// TwinCAT 3 PLC project PLC1
// ProgramVersion: 3.1.4024.0
// libraries:
//   Tc2_Standard, * (Beckhoff Automation GmbH)
//   Tc2_System, * (Beckhoff Automation GmbH)
//   Tc3_Module, * (Beckhoff Automation GmbH)
// project tree:
//   / PlcTask.TcTTO
//   POUs/ FB_ParseString.TcPOU, MAIN.TcPOU
// real-time tasks:
//   TASK PlcTask: cycle T#10ms, priority 20, ADS port 350

CONFIGURATION PLC1
    RESOURCE PLC ON TwinCAT3
        TASK PlcTask(INTERVAL := T#10ms, PRIORITY := 20);
        PROGRAM MAIN WITH PlcTask : MAIN;
    END_RESOURCE
END_CONFIGURATION

// ---- POUs/MAIN.TcPOU
PROGRAM MAIN
VAR
END_VAR

END_PROGRAM

// ---- POUs/FB_ParseString.TcPOU
FUNCTION_BLOCK FB_ParseString
VAR_INPUT
	sCharToSearch : STRING;
	sInputString  : STRING;
END_VAR
VAR_OUTPUT
	sStringParsed : STRING;
END_VAR
VAR
	Position: INT;
END_VAR

Position := FIND(sInputString, sCharToSearch);
sStringParsed := DELETE(sInputString, Position, LEN(sInputString));

END_FUNCTION_BLOCK
